{attribute 'GeneratedUsingTerminal: EK1122-0000-0018'}
{attribute addProperty BoxType "EK1122-0000-0018"}
{attribute addProperty Id "Beckhoff_ER2xxxsub_EK1100EK1100_1FC0878B2A_0001_ER2008_0001_0018ER2008_E2806B9511A_0002_ER2008_0001_0019ER2008_E2806B9511A_0003_ER2008_0002_0018ER2008_E2806B9511A_0004_ER2008_0002_0019ER2008_E2806B9511A_0005_ER2008_0022_0017ER2008_E2806B9511A_0006_ER2008_0022_0018ER2008_E2806B9511A_0007_ER2028_0001_0017ER2028_E2806B9511A_0008_ER2028_0001_0018ER2028_E2806B9511A_0009_ER2028_0002_0018ER2028_E2806B9511A_0010_ER2028_0002_0019ER2028_E2806B9511A_0011_ER2028_1032_0016ER2028_E2806B9511A_0012_ER2038_0001_0017ER2038_3AE10DD720A_0013_ER2038_0001_0018ER2038_3AE10DD720A_0014_ER2038_0002_0017ER2038_3AE10DD720A_0015_ER2038_0002_0018ER2038_3AE10DD720A_0016_ER2308_0001_0018ER2308_F6D9A8D112A_0017_ER2308_0001_0019ER2308_F6D9A8D112A_0018_ER2308_0002_0018ER2308_F6D9A8D112A_0019_ER2308_0002_0019ER2308_F6D9A8D112A_0020_ER2318_0001_0018ER2318_F6D9A8D112A_0021_ER2318_0001_0019ER2318_F6D9A8D112A_0022_ER2318_0002_0018ER2318_F6D9A8D112A_0023_ER2318_0002_0019ER2318_F6D9A8D112A_0024_ER2328_0001_0017ER2328_F6D9A8D112A_0025_ER2328_0001_0018ER2328_F6D9A8D112A_0026_ER2328_0002_0018ER2328_F6D9A8D112A_0027_ER2328_0002_0019ER2328_F6D9A8D112A_0028_ER2338_0001_0022ER2338_7699BCF620A_0029_ER2338_0001_0023ER2338_7699BCF620A_0030_ER2338_0002_0022ER2338_7699BCF620A_0031_ER2338_0002_0023ER2338_7699BCF620A_0032_ER2338_1001_0017ER2338_7699BCF620A_0033_ER2338_1001_0018ER2338_7699BCF620A_0034_ER2338_1002_0017ER2338_7699BCF620A_0035_ER2338_1002_0018ER2338_7699BCF620A_0036_ER2339_0021_0018ER2339_6DDDF9AF36A_0037_ER2339_0021_0019ER2339_4CF33DED36A_0038_ER2339_0022_0018ER2339_4CF33DED36A_0039_ER2339_0022_0019ER2339_4CF33DED36A_0040_ER2349_0021_0017ER2349_4CF33DED36A_0041_ER2349_0021_0018ER2349_4CF33DED36A_0042_ER2349_0022_0017ER2349_4CF33DED36A_0043_ER2349_0022_0018ER2349_4CF33DED36A_0044_ER2624_0002_0018ER2624_7B64371E7A_0045_ER2624_0002_0019ER2624_7B64371E7A_0046_ER2809_0021_0017ER2809_2B6483BD19A_0047_ER2809_0021_0018ER2809_2B6483BD19A_0048_ER2809_0022_0016ER2809_2B6483BD19A_0049_ER2809_0022_0017ER2809_2B6483BD19A_0050_ER2809_0022_0018ER2809_2B6483BD19"}
{attribute addProperty CRC "3887409694"}
{attribute addProperty Size "904"}
TYPE Beckhoff_ER2xxxEK1122_E7B52A1E EXTENDS EK1122_1FC0878B :
STRUCT
	{attribute addProperty Name "Beckhoff_ER2xxxsub_EK1100"}
	{attribute addProperty PreviousPort "Beckhoff ER2xxxEK1122 : D"}
	Beckhoff_ER2xxxsub_EK1100 : EK1100_1FC0878B;
	{attribute addProperty Name "A_0001_ER2008_0001_0018"}
	{attribute addProperty PreviousPort "Beckhoff ER2xxxsub EK1100 : C"}
	A_0001_ER2008_0001_0018 : ER2008_E2806B95;
	{attribute addProperty Name "A_0002_ER2008_0001_0019"}
	{attribute addProperty PreviousPort "A_0001(ER2008-0001-0018) : B"}
	A_0002_ER2008_0001_0019 : ER2008_E2806B95;
	{attribute addProperty Name "A_0003_ER2008_0002_0018"}
	{attribute addProperty PreviousPort "A_0002(ER2008-0001-0019) : B"}
	A_0003_ER2008_0002_0018 : ER2008_E2806B95;
	{attribute addProperty Name "A_0004_ER2008_0002_0019"}
	{attribute addProperty PreviousPort "A_0003(ER2008-0002-0018) : B"}
	A_0004_ER2008_0002_0019 : ER2008_E2806B95;
	{attribute addProperty Name "A_0005_ER2008_0022_0017"}
	{attribute addProperty PreviousPort "A_0004(ER2008-0002-0019) : B"}
	A_0005_ER2008_0022_0017 : ER2008_E2806B95;
	{attribute addProperty Name "A_0006_ER2008_0022_0018"}
	{attribute addProperty PreviousPort "A_0005(ER2008-0022-0017) : B"}
	A_0006_ER2008_0022_0018 : ER2008_E2806B95;
	{attribute addProperty Name "A_0007_ER2028_0001_0017"}
	{attribute addProperty PreviousPort "A_0006(ER2008-0022-0018) : B"}
	A_0007_ER2028_0001_0017 : ER2028_E2806B95;
	{attribute addProperty Name "A_0008_ER2028_0001_0018"}
	{attribute addProperty PreviousPort "A_0007(ER2028-0001-0017) : B"}
	A_0008_ER2028_0001_0018 : ER2028_E2806B95;
	{attribute addProperty Name "A_0009_ER2028_0002_0018"}
	{attribute addProperty PreviousPort "A_0008(ER2028-0001-0018) : B"}
	A_0009_ER2028_0002_0018 : ER2028_E2806B95;
	{attribute addProperty Name "A_0010_ER2028_0002_0019"}
	{attribute addProperty PreviousPort "A_0009(ER2028-0002-0018) : B"}
	A_0010_ER2028_0002_0019 : ER2028_E2806B95;
	{attribute addProperty Name "A_0011_ER2028_1032_0016"}
	{attribute addProperty PreviousPort "A_0010(ER2028-0002-0019) : B"}
	A_0011_ER2028_1032_0016 : ER2028_E2806B95;
	{attribute addProperty Name "A_0012_ER2038_0001_0017"}
	{attribute addProperty PreviousPort "A_0011(ER2028-1032-0016) : B"}
	A_0012_ER2038_0001_0017 : ER2038_3AE10DD7;
	{attribute addProperty Name "A_0013_ER2038_0001_0018"}
	{attribute addProperty PreviousPort "A_0012(ER2038-0001-0017) : B"}
	A_0013_ER2038_0001_0018 : ER2038_3AE10DD7;
	{attribute addProperty Name "A_0014_ER2038_0002_0017"}
	{attribute addProperty PreviousPort "A_0013(ER2038-0001-0018) : B"}
	A_0014_ER2038_0002_0017 : ER2038_3AE10DD7;
	{attribute addProperty Name "A_0015_ER2038_0002_0018"}
	{attribute addProperty PreviousPort "A_0014(ER2038-0002-0017) : B"}
	A_0015_ER2038_0002_0018 : ER2038_3AE10DD7;
	{attribute addProperty Name "A_0016_ER2308_0001_0018"}
	{attribute addProperty PreviousPort "A_0015(ER2038-0002-0018) : B"}
	A_0016_ER2308_0001_0018 : ER2308_F6D9A8D1;
	{attribute addProperty Name "A_0017_ER2308_0001_0019"}
	{attribute addProperty PreviousPort "A_0016(ER2308-0001-0018) : B"}
	A_0017_ER2308_0001_0019 : ER2308_F6D9A8D1;
	{attribute addProperty Name "A_0018_ER2308_0002_0018"}
	{attribute addProperty PreviousPort "A_0017(ER2308-0001-0019) : B"}
	A_0018_ER2308_0002_0018 : ER2308_F6D9A8D1;
	{attribute addProperty Name "A_0019_ER2308_0002_0019"}
	{attribute addProperty PreviousPort "A_0018(ER2308-0002-0018) : B"}
	A_0019_ER2308_0002_0019 : ER2308_F6D9A8D1;
	{attribute addProperty Name "A_0020_ER2318_0001_0018"}
	{attribute addProperty PreviousPort "A_0019(ER2308-0002-0019) : B"}
	A_0020_ER2318_0001_0018 : ER2318_F6D9A8D1;
	{attribute addProperty Name "A_0021_ER2318_0001_0019"}
	{attribute addProperty PreviousPort "A_0020(ER2318-0001-0018) : B"}
	A_0021_ER2318_0001_0019 : ER2318_F6D9A8D1;
	{attribute addProperty Name "A_0022_ER2318_0002_0018"}
	{attribute addProperty PreviousPort "A_0021(ER2318-0001-0019) : B"}
	A_0022_ER2318_0002_0018 : ER2318_F6D9A8D1;
	{attribute addProperty Name "A_0023_ER2318_0002_0019"}
	{attribute addProperty PreviousPort "A_0022(ER2318-0002-0018) : B"}
	A_0023_ER2318_0002_0019 : ER2318_F6D9A8D1;
	{attribute addProperty Name "A_0024_ER2328_0001_0017"}
	{attribute addProperty PreviousPort "A_0023(ER2318-0002-0019) : B"}
	A_0024_ER2328_0001_0017 : ER2328_F6D9A8D1;
	{attribute addProperty Name "A_0025_ER2328_0001_0018"}
	{attribute addProperty PreviousPort "A_0024(ER2328-0001-0017) : B"}
	A_0025_ER2328_0001_0018 : ER2328_F6D9A8D1;
	{attribute addProperty Name "A_0026_ER2328_0002_0018"}
	{attribute addProperty PreviousPort "A_0025(ER2328-0001-0018) : B"}
	A_0026_ER2328_0002_0018 : ER2328_F6D9A8D1;
	{attribute addProperty Name "A_0027_ER2328_0002_0019"}
	{attribute addProperty PreviousPort "A_0026(ER2328-0002-0018) : B"}
	A_0027_ER2328_0002_0019 : ER2328_F6D9A8D1;
	{attribute addProperty Name "A_0028_ER2338_0001_0022"}
	{attribute addProperty PreviousPort "A_0027(ER2328-0002-0019) : B"}
	A_0028_ER2338_0001_0022 : ER2338_7699BCF6;
	{attribute addProperty Name "A_0029_ER2338_0001_0023"}
	{attribute addProperty PreviousPort "A_0028(ER2338-0001-0022) : B"}
	A_0029_ER2338_0001_0023 : ER2338_7699BCF6;
	{attribute addProperty Name "A_0030_ER2338_0002_0022"}
	{attribute addProperty PreviousPort "A_0029(ER2338-0001-0023) : B"}
	A_0030_ER2338_0002_0022 : ER2338_7699BCF6;
	{attribute addProperty Name "A_0031_ER2338_0002_0023"}
	{attribute addProperty PreviousPort "A_0030(ER2338-0002-0022) : B"}
	A_0031_ER2338_0002_0023 : ER2338_7699BCF6;
	{attribute addProperty Name "A_0032_ER2338_1001_0017"}
	{attribute addProperty PreviousPort "A_0031(ER2338-0002-0023) : B"}
	A_0032_ER2338_1001_0017 : ER2338_7699BCF6;
	{attribute addProperty Name "A_0033_ER2338_1001_0018"}
	{attribute addProperty PreviousPort "A_0032(ER2338-1001-0017) : B"}
	A_0033_ER2338_1001_0018 : ER2338_7699BCF6;
	{attribute addProperty Name "A_0034_ER2338_1002_0017"}
	{attribute addProperty PreviousPort "A_0033(ER2338-1001-0018) : B"}
	A_0034_ER2338_1002_0017 : ER2338_7699BCF6;
	{attribute addProperty Name "A_0035_ER2338_1002_0018"}
	{attribute addProperty PreviousPort "A_0034(ER2338-1002-0017) : B"}
	A_0035_ER2338_1002_0018 : ER2338_7699BCF6;
	{attribute addProperty Name "A_0036_ER2339_0021_0018"}
	{attribute addProperty PreviousPort "A_0035(ER2338-1002-0018) : B"}
	A_0036_ER2339_0021_0018 : ER2339_6DDDF9AF;
	{attribute addProperty Name "A_0037_ER2339_0021_0019"}
	{attribute addProperty PreviousPort "A_0036(ER2339-0021-0018) : B"}
	A_0037_ER2339_0021_0019 : ER2339_4CF33DED;
	{attribute addProperty Name "A_0038_ER2339_0022_0018"}
	{attribute addProperty PreviousPort "A_0037(ER2339-0021-0019) : B"}
	A_0038_ER2339_0022_0018 : ER2339_4CF33DED;
	{attribute addProperty Name "A_0039_ER2339_0022_0019"}
	{attribute addProperty PreviousPort "A_0038(ER2339-0022-0018) : B"}
	A_0039_ER2339_0022_0019 : ER2339_4CF33DED;
	{attribute addProperty Name "A_0040_ER2349_0021_0017"}
	{attribute addProperty PreviousPort "A_0039(ER2339-0022-0019) : B"}
	A_0040_ER2349_0021_0017 : ER2349_4CF33DED;
	{attribute addProperty Name "A_0041_ER2349_0021_0018"}
	{attribute addProperty PreviousPort "A_0040(ER2349-0021-0017) : B"}
	A_0041_ER2349_0021_0018 : ER2349_4CF33DED;
	{attribute addProperty Name "A_0042_ER2349_0022_0017"}
	{attribute addProperty PreviousPort "A_0041(ER2349-0021-0018) : B"}
	A_0042_ER2349_0022_0017 : ER2349_4CF33DED;
	{attribute addProperty Name "A_0043_ER2349_0022_0018"}
	{attribute addProperty PreviousPort "A_0042(ER2349-0022-0017) : B"}
	A_0043_ER2349_0022_0018 : ER2349_4CF33DED;
	{attribute addProperty Name "A_0044_ER2624_0002_0018"}
	{attribute addProperty PreviousPort "A_0043(ER2349-0022-0018) : B"}
	A_0044_ER2624_0002_0018 : ER2624_7B64371E;
	{attribute addProperty Name "A_0045_ER2624_0002_0019"}
	{attribute addProperty PreviousPort "A_0044(ER2624-0002-0018) : B"}
	A_0045_ER2624_0002_0019 : ER2624_7B64371E;
	{attribute addProperty Name "A_0046_ER2809_0021_0017"}
	{attribute addProperty PreviousPort "A_0045(ER2624-0002-0019) : B"}
	A_0046_ER2809_0021_0017 : ER2809_2B6483BD;
	{attribute addProperty Name "A_0047_ER2809_0021_0018"}
	{attribute addProperty PreviousPort "A_0046(ER2809-0021-0017) : B"}
	A_0047_ER2809_0021_0018 : ER2809_2B6483BD;
	{attribute addProperty Name "A_0048_ER2809_0022_0016"}
	{attribute addProperty PreviousPort "A_0047(ER2809-0021-0018) : B"}
	A_0048_ER2809_0022_0016 : ER2809_2B6483BD;
	{attribute addProperty Name "A_0049_ER2809_0022_0017"}
	{attribute addProperty PreviousPort "A_0048(ER2809-0022-0016) : B"}
	A_0049_ER2809_0022_0017 : ER2809_2B6483BD;
	{attribute addProperty Name "A_0050_ER2809_0022_0018"}
	{attribute addProperty PreviousPort "A_0049(ER2809-0022-0017) : B"}
	A_0050_ER2809_0022_0018 : ER2809_2B6483BD;
END_STRUCT
END_TYPE

(* stored: Version 1.2.0.0, ProductVersion 3.1.4024.9
   DUT Beckhoff_ER2xxxEK1122_E7B52A1E: Id {867bb656-cfce-4d32-891e-b7c2eaebf547} *)
